// TIA Portal V17 export
// export: Created 2023-02-14T02:49:31.6771521Z, ExportSetting WithDefaults, DisplayName Totally Integrated Automation Portal, DisplayVersion V17, DisplayName TIA Portal Openness, DisplayVersion V17, DisplayName TIA Portal Teamcenter Gateway, DisplayVersion V17, DisplayName TIA Portal Version Control Interface, DisplayVersion V17, DisplayName SINAMICS Startdrive Advanced, DisplayVersion V17, DisplayName SINAMICS Startdrive G130, G150, S120, S150, SINAMICS MV, S210, DisplayVersion V17, DisplayName SINAMICS Startdrive G110M, G120, G120C, G120D, G120P, G115D, DisplayVersion V17, DisplayName STEP 7 Professional, DisplayVersion V17, DisplayName STEP 7 Safety, DisplayVersion V17, DisplayName WinCC Professional, DisplayVersion V17
FUNCTION_BLOCK "IO Motor MCC Preparation"   // FB15, LAD
{ S7_Optimized_Access := 'FALSE' }
VERSION : 0.1
// stored: AutoNumber true, IsIECCheckEnabled false, SetENOAutomatically false, UDAEnableTagReadback false
   VAR_INPUT
      lock : Bool;
      Init : Bool;
      EM_Stop : Bool;
      Testing : Bool;
      Reset : Bool;
   END_VAR
   VAR
      "P-01.01" { S7_SetPoint := 'True'} : "Motor_w_VSD";
      "P-02.01" { S7_SetPoint := 'True'} : "Motor_w_VSD";
      "P-02.03" { S7_SetPoint := 'True'} : "Motor_w_VSD";
      "P-03.01" { S7_SetPoint := 'True'} : "Motor_w_VSD";
      "P-03.03" { S7_SetPoint := 'True'} : "Motor_w_VSD";
      "P-04.01" { S7_SetPoint := 'True'} : "Motor_w_VSD";
      "XA-05.01" { S7_SetPoint := 'True'} : "Motor_w_VSD";
      "P-05.01" { S7_SetPoint := 'True'} : "Motor_w_VSD";
      "P-05.03_DOL" { S7_SetPoint := 'True'} : "Motor";
      "P-06.01" { S7_SetPoint := 'True'} : "Motor_w_VSD";
      "P-07.01" { S7_SetPoint := 'True'} : "Motor_w_VSD";
      "P-08.01" { S7_SetPoint := 'True'} : "Motor_w_VSD";
      "P-08.02" { S7_SetPoint := 'True'} : "Motor_w_VSD";
      "XA-09.01" { S7_SetPoint := 'True'} : "Motor_w_VSD";
      "P-09.01" { S7_SetPoint := 'True'} : "Motor_w_VSD";
      "P-09.03" { S7_SetPoint := 'True'} : "Motor";
      "P-10.01" { S7_SetPoint := 'True'} : "Motor_w_VSD";
      "P-51.01" { S7_SetPoint := 'True'} : "Motor_w_VSD";
   END_VAR
BEGIN

REGION Network 1: Testing
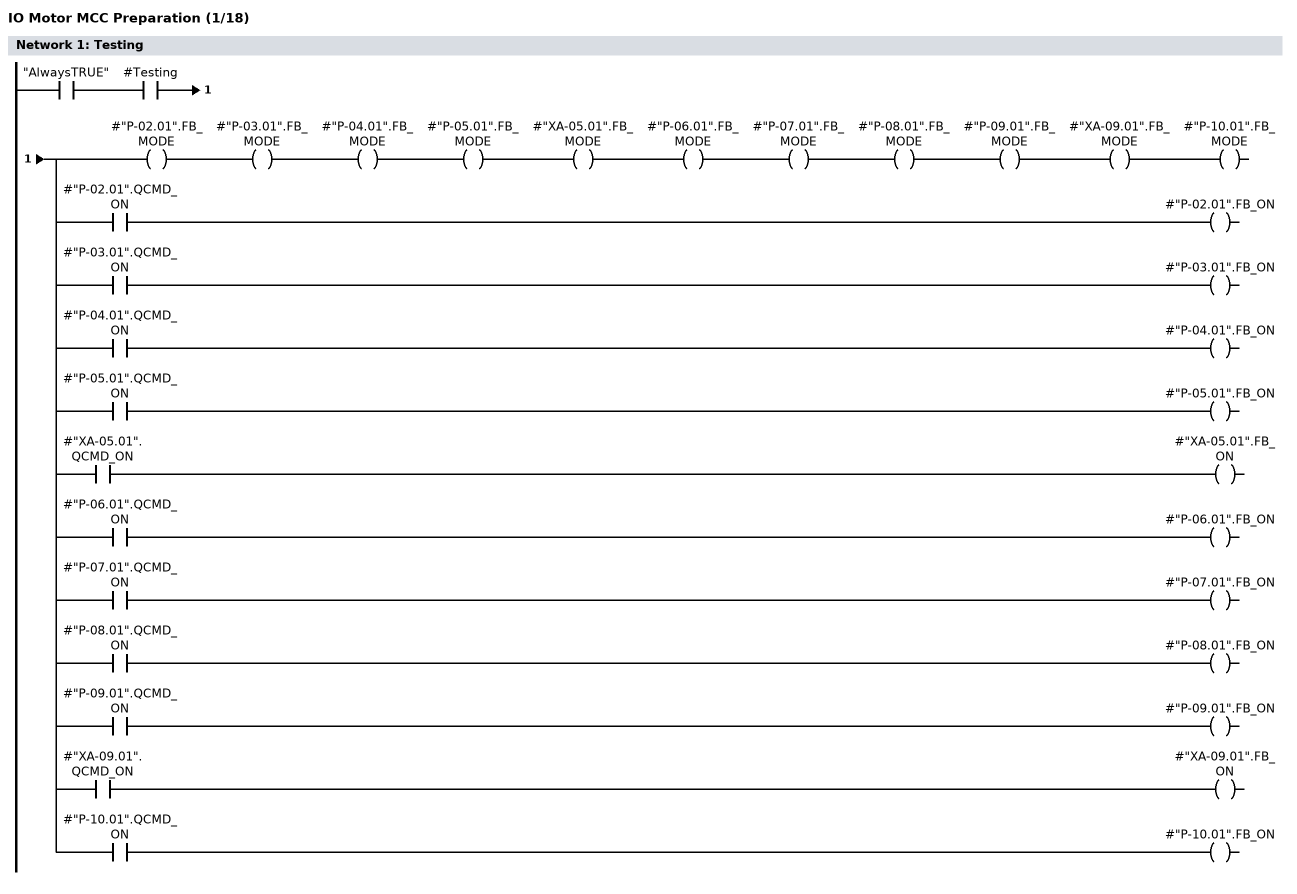
   RUNG wire#powerrail
      Contact( "AlwaysTRUE" )
      Contact( #Testing )
      wire#w1
      Coil( #"P-02.01".FB_MODE )
      Coil( #"P-03.01".FB_MODE )
      Coil( #"P-04.01".FB_MODE )
      Coil( #"P-05.01".FB_MODE )
      Coil( #"XA-05.01".FB_MODE )
      Coil( #"P-06.01".FB_MODE )
      Coil( #"P-07.01".FB_MODE )
      Coil( #"P-08.01".FB_MODE )
      Coil( #"P-09.01".FB_MODE )
      Coil( #"XA-09.01".FB_MODE )
      Coil( #"P-10.01".FB_MODE )
   END_RUNG
   RUNG wire#w1
      Contact( #"P-02.01".QCMD_ON )
      Coil( #"P-02.01".FB_ON )
   END_RUNG
   RUNG wire#w1
      Contact( #"P-03.01".QCMD_ON )
      Coil( #"P-03.01".FB_ON )
   END_RUNG
   RUNG wire#w1
      Contact( #"P-04.01".QCMD_ON )
      Coil( #"P-04.01".FB_ON )
   END_RUNG
   RUNG wire#w1
      Contact( #"P-05.01".QCMD_ON )
      Coil( #"P-05.01".FB_ON )
   END_RUNG
   RUNG wire#w1
      Contact( #"XA-05.01".QCMD_ON )
      Coil( #"XA-05.01".FB_ON )
   END_RUNG
   RUNG wire#w1
      Contact( #"P-06.01".QCMD_ON )
      Coil( #"P-06.01".FB_ON )
   END_RUNG
   RUNG wire#w1
      Contact( #"P-07.01".QCMD_ON )
      Coil( #"P-07.01".FB_ON )
   END_RUNG
   RUNG wire#w1
      Contact( #"P-08.01".QCMD_ON )
      Coil( #"P-08.01".FB_ON )
   END_RUNG
   RUNG wire#w1
      Contact( #"P-09.01".QCMD_ON )
      Coil( #"P-09.01".FB_ON )
   END_RUNG
   RUNG wire#w1
      Contact( #"XA-09.01".QCMD_ON )
      Coil( #"XA-09.01".FB_ON )
   END_RUNG
   RUNG wire#w1
      Contact( #"P-10.01".QCMD_ON )
      Coil( #"P-10.01".FB_ON )
   END_RUNG
   // the same network as SCL:
   #"P-02.01".FB_MODE := "AlwaysTRUE" AND #Testing;
   #"P-03.01".FB_MODE := #"P-02.01".FB_MODE;
   #"P-04.01".FB_MODE := #"P-02.01".FB_MODE;
   #"P-05.01".FB_MODE := #"P-02.01".FB_MODE;
   #"XA-05.01".FB_MODE := #"P-02.01".FB_MODE;
   #"P-06.01".FB_MODE := #"P-02.01".FB_MODE;
   #"P-07.01".FB_MODE := #"P-02.01".FB_MODE;
   #"P-08.01".FB_MODE := #"P-02.01".FB_MODE;
   #"P-09.01".FB_MODE := #"P-02.01".FB_MODE;
   #"XA-09.01".FB_MODE := #"P-02.01".FB_MODE;
   #"P-10.01".FB_MODE := #"P-02.01".FB_MODE;
   #"P-02.01".FB_ON := #"P-02.01".FB_MODE AND #"P-02.01".QCMD_ON;
   #"P-03.01".FB_ON := #"P-02.01".FB_MODE AND #"P-03.01".QCMD_ON;
   #"P-04.01".FB_ON := #"P-02.01".FB_MODE AND #"P-04.01".QCMD_ON;
   #"P-05.01".FB_ON := #"P-02.01".FB_MODE AND #"P-05.01".QCMD_ON;
   #"XA-05.01".FB_ON := #"P-02.01".FB_MODE AND #"XA-05.01".QCMD_ON;
   #"P-06.01".FB_ON := #"P-02.01".FB_MODE AND #"P-06.01".QCMD_ON;
   #"P-07.01".FB_ON := #"P-02.01".FB_MODE AND #"P-07.01".QCMD_ON;
   #"P-08.01".FB_ON := #"P-02.01".FB_MODE AND #"P-08.01".QCMD_ON;
   #"P-09.01".FB_ON := #"P-02.01".FB_MODE AND #"P-09.01".QCMD_ON;
   #"XA-09.01".FB_ON := #"P-02.01".FB_MODE AND #"XA-09.01".QCMD_ON;
   #"P-10.01".FB_ON := #"P-02.01".FB_MODE AND #"P-10.01".QCMD_ON;
END_REGION

REGION Network 2: P-02.01
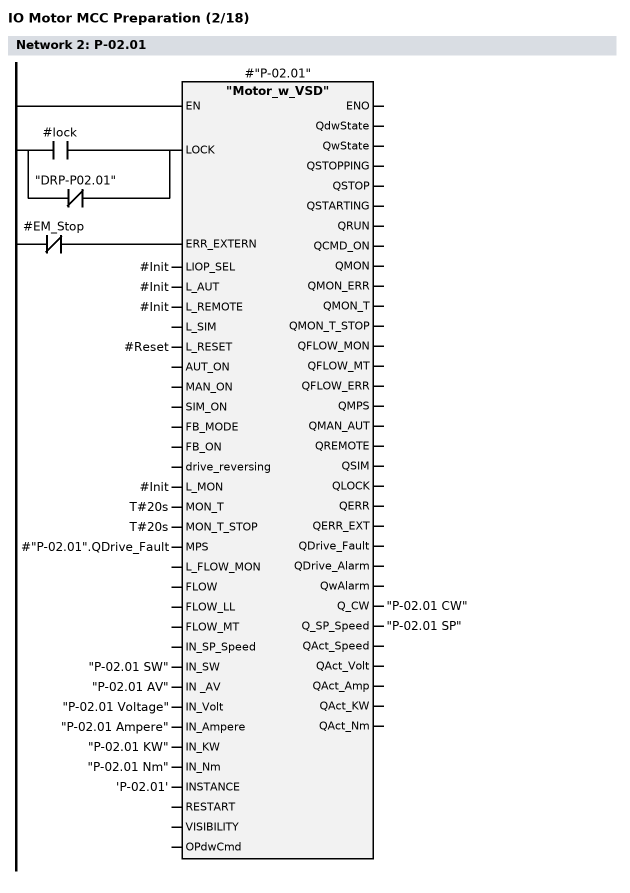
   RUNG wire#powerrail
      #"P-02.01"(LOCK := wire#w1, ERR_EXTERN := wire#w2, LIOP_SEL := #Init, L_AUT := #Init, L_REMOTE := #Init, L_SIM :=, L_RESET := #Reset, AUT_ON :=, MAN_ON :=, SIM_ON :=, FB_MODE :=, FB_ON :=, drive_reversing :=, L_MON := #Init, MON_T := T#20s, MON_T_STOP := T#20s, MPS := #"P-02.01".QDrive_Fault, L_FLOW_MON :=, FLOW :=, FLOW_LL :=, FLOW_MT :=, IN_SP_Speed :=, IN_SW := "P-02.01 SW", "IN _AV" := "P-02.01 AV", IN_Volt := "P-02.01 Voltage", IN_Ampere := "P-02.01 Ampere", IN_KW := "P-02.01 KW", IN_Nm := "P-02.01 Nm", INSTANCE := 'P-02.01', RESTART :=, VISIBILITY :=, OPdwCmd :=, QdwState =>, QwState =>, QSTOPPING =>, QSTOP =>, QSTARTING =>, QRUN =>, QCMD_ON =>, QMON =>, QMON_ERR =>, QMON_T =>, QMON_T_STOP =>, QFLOW_MON =>, QFLOW_MT =>, QFLOW_ERR =>, QMPS =>, QMAN_AUT =>, QREMOTE =>, QSIM =>, QLOCK =>, QERR =>, QERR_EXT =>, QDrive_Fault =>, QDrive_Alarm =>, QwAlarm =>, Q_CW => "P-02.01 CW", Q_SP_Speed => "P-02.01 SP", QAct_Speed =>, QAct_Volt =>, QAct_Amp =>, QAct_KW =>, QAct_Nm =>)
   END_RUNG
   RUNG wire#powerrail
      Contact( #lock )
   END_RUNG wire#w1
   RUNG wire#powerrail
      I_Contact( "DRP-P02.01" )
   END_RUNG wire#w1
   RUNG wire#powerrail
      I_Contact( #EM_Stop )
   END_RUNG wire#w2
   // the same network as SCL:
   #"P-02.01"(LOCK := #lock OR NOT "DRP-P02.01",   // "Motor_w_VSD"
              ERR_EXTERN := NOT #EM_Stop,
              LIOP_SEL := #Init,
              L_AUT := #Init,
              L_REMOTE := #Init,
              L_RESET := #Reset,
              L_MON := #Init,
              MON_T := T#20s,
              MON_T_STOP := T#20s,
              MPS := #"P-02.01".QDrive_Fault,
              IN_SW := "P-02.01 SW",
              "IN _AV" := "P-02.01 AV",
              IN_Volt := "P-02.01 Voltage",
              IN_Ampere := "P-02.01 Ampere",
              IN_KW := "P-02.01 KW",
              IN_Nm := "P-02.01 Nm",
              INSTANCE := 'P-02.01',
              Q_CW => "P-02.01 CW",
              Q_SP_Speed => "P-02.01 SP");
END_REGION

REGION Network 3: P-02.03
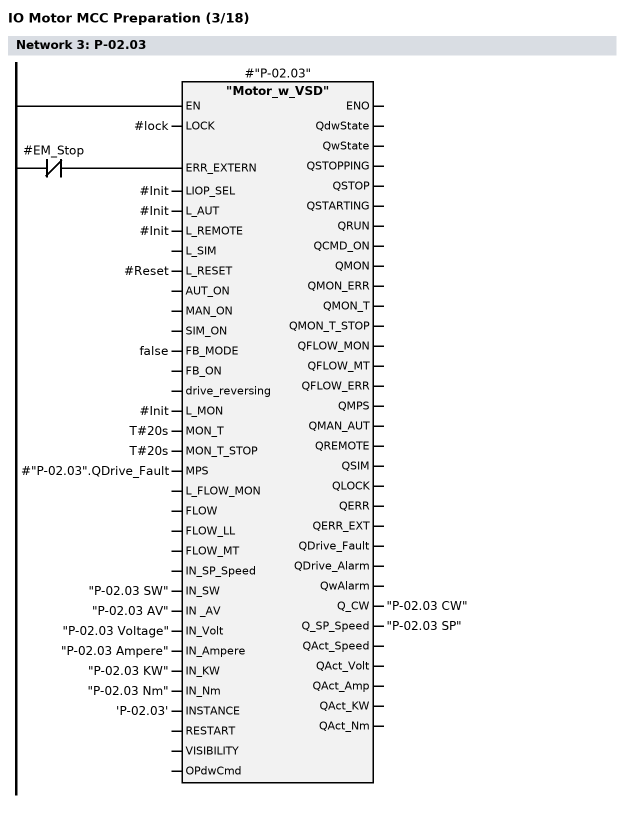
   RUNG wire#powerrail
      #"P-02.03"(ERR_EXTERN := wire#w1, LOCK := #lock, LIOP_SEL := #Init, L_AUT := #Init, L_REMOTE := #Init, L_SIM :=, L_RESET := #Reset, AUT_ON :=, MAN_ON :=, SIM_ON :=, FB_MODE := false, FB_ON :=, drive_reversing :=, L_MON := #Init, MON_T := T#20s, MON_T_STOP := T#20s, MPS := #"P-02.03".QDrive_Fault, L_FLOW_MON :=, FLOW :=, FLOW_LL :=, FLOW_MT :=, IN_SP_Speed :=, IN_SW := "P-02.03 SW", "IN _AV" := "P-02.03 AV", IN_Volt := "P-02.03 Voltage", IN_Ampere := "P-02.03 Ampere", IN_KW := "P-02.03 KW", IN_Nm := "P-02.03 Nm", INSTANCE := 'P-02.03', RESTART :=, VISIBILITY :=, OPdwCmd :=, QdwState =>, QwState =>, QSTOPPING =>, QSTOP =>, QSTARTING =>, QRUN =>, QCMD_ON =>, QMON =>, QMON_ERR =>, QMON_T =>, QMON_T_STOP =>, QFLOW_MON =>, QFLOW_MT =>, QFLOW_ERR =>, QMPS =>, QMAN_AUT =>, QREMOTE =>, QSIM =>, QLOCK =>, QERR =>, QERR_EXT =>, QDrive_Fault =>, QDrive_Alarm =>, QwAlarm =>, Q_CW => "P-02.03 CW", Q_SP_Speed => "P-02.03 SP", QAct_Speed =>, QAct_Volt =>, QAct_Amp =>, QAct_KW =>, QAct_Nm =>)
   END_RUNG
   RUNG wire#powerrail
      I_Contact( #EM_Stop )
   END_RUNG wire#w1
   // the same network as SCL:
   #"P-02.03"(LOCK := #lock,   // "Motor_w_VSD"
              ERR_EXTERN := NOT #EM_Stop,
              LIOP_SEL := #Init,
              L_AUT := #Init,
              L_REMOTE := #Init,
              L_RESET := #Reset,
              FB_MODE := false,
              L_MON := #Init,
              MON_T := T#20s,
              MON_T_STOP := T#20s,
              MPS := #"P-02.03".QDrive_Fault,
              IN_SW := "P-02.03 SW",
              "IN _AV" := "P-02.03 AV",
              IN_Volt := "P-02.03 Voltage",
              IN_Ampere := "P-02.03 Ampere",
              IN_KW := "P-02.03 KW",
              IN_Nm := "P-02.03 Nm",
              INSTANCE := 'P-02.03',
              Q_CW => "P-02.03 CW",
              Q_SP_Speed => "P-02.03 SP");
END_REGION

REGION Network 4: P-03.01
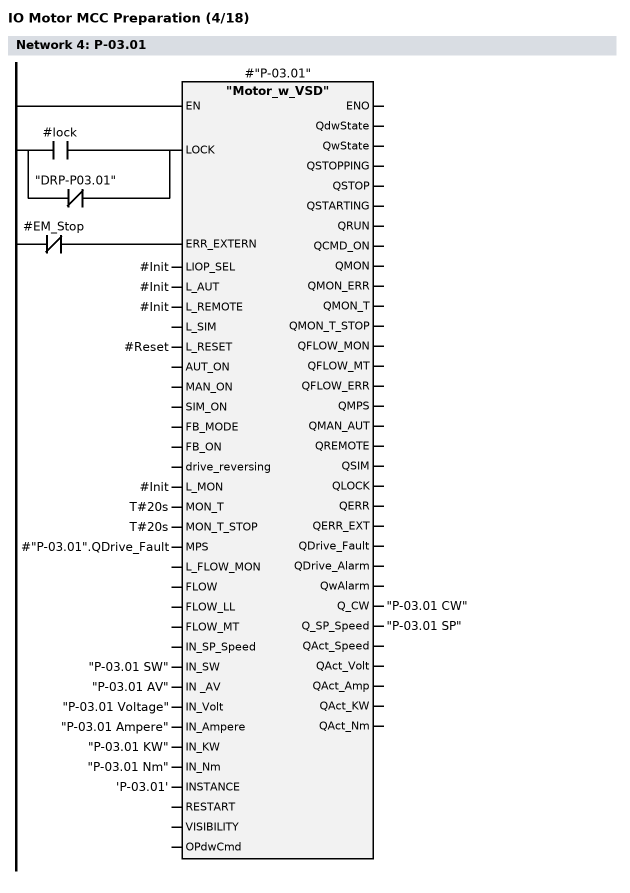
   RUNG wire#powerrail
      #"P-03.01"(LOCK := wire#w1, ERR_EXTERN := wire#w2, LIOP_SEL := #Init, L_AUT := #Init, L_REMOTE := #Init, L_SIM :=, L_RESET := #Reset, AUT_ON :=, MAN_ON :=, SIM_ON :=, FB_MODE :=, FB_ON :=, drive_reversing :=, L_MON := #Init, MON_T := T#20s, MON_T_STOP := T#20s, MPS := #"P-03.01".QDrive_Fault, L_FLOW_MON :=, FLOW :=, FLOW_LL :=, FLOW_MT :=, IN_SP_Speed :=, IN_SW := "P-03.01 SW", "IN _AV" := "P-03.01 AV", IN_Volt := "P-03.01 Voltage", IN_Ampere := "P-03.01 Ampere", IN_KW := "P-03.01 KW", IN_Nm := "P-03.01 Nm", INSTANCE := 'P-03.01', RESTART :=, VISIBILITY :=, OPdwCmd :=, QdwState =>, QwState =>, QSTOPPING =>, QSTOP =>, QSTARTING =>, QRUN =>, QCMD_ON =>, QMON =>, QMON_ERR =>, QMON_T =>, QMON_T_STOP =>, QFLOW_MON =>, QFLOW_MT =>, QFLOW_ERR =>, QMPS =>, QMAN_AUT =>, QREMOTE =>, QSIM =>, QLOCK =>, QERR =>, QERR_EXT =>, QDrive_Fault =>, QDrive_Alarm =>, QwAlarm =>, Q_CW => "P-03.01 CW", Q_SP_Speed => "P-03.01 SP", QAct_Speed =>, QAct_Volt =>, QAct_Amp =>, QAct_KW =>, QAct_Nm =>)
   END_RUNG
   RUNG wire#powerrail
      Contact( #lock )
   END_RUNG wire#w1
   RUNG wire#powerrail
      I_Contact( "DRP-P03.01" )
   END_RUNG wire#w1
   RUNG wire#powerrail
      I_Contact( #EM_Stop )
   END_RUNG wire#w2
   // the same network as SCL:
   #"P-03.01"(LOCK := #lock OR NOT "DRP-P03.01",   // "Motor_w_VSD"
              ERR_EXTERN := NOT #EM_Stop,
              LIOP_SEL := #Init,
              L_AUT := #Init,
              L_REMOTE := #Init,
              L_RESET := #Reset,
              L_MON := #Init,
              MON_T := T#20s,
              MON_T_STOP := T#20s,
              MPS := #"P-03.01".QDrive_Fault,
              IN_SW := "P-03.01 SW",
              "IN _AV" := "P-03.01 AV",
              IN_Volt := "P-03.01 Voltage",
              IN_Ampere := "P-03.01 Ampere",
              IN_KW := "P-03.01 KW",
              IN_Nm := "P-03.01 Nm",
              INSTANCE := 'P-03.01',
              Q_CW => "P-03.01 CW",
              Q_SP_Speed => "P-03.01 SP");
END_REGION

REGION Network 5: P-03.03
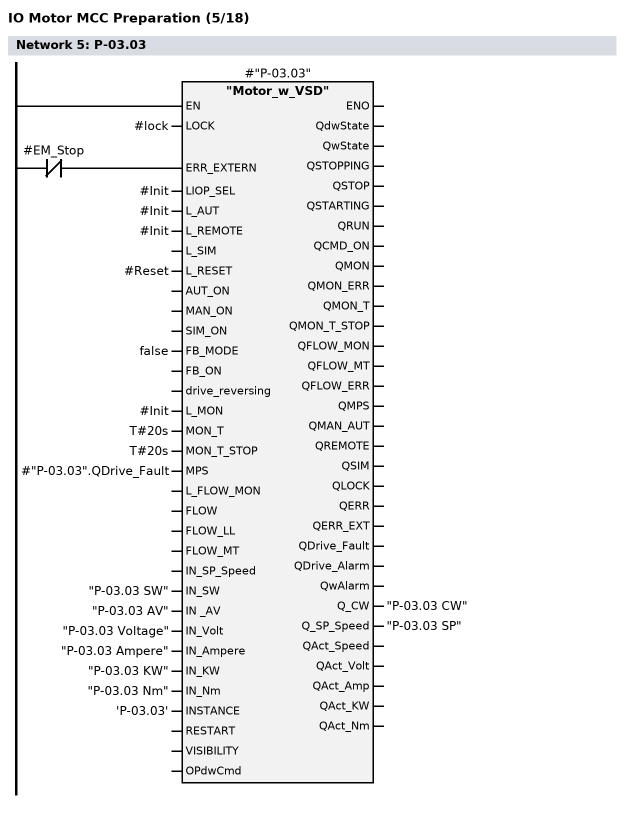
   RUNG wire#powerrail
      #"P-03.03"(ERR_EXTERN := wire#w1, LOCK := #lock, LIOP_SEL := #Init, L_AUT := #Init, L_REMOTE := #Init, L_SIM :=, L_RESET := #Reset, AUT_ON :=, MAN_ON :=, SIM_ON :=, FB_MODE := false, FB_ON :=, drive_reversing :=, L_MON := #Init, MON_T := T#20s, MON_T_STOP := T#20s, MPS := #"P-03.03".QDrive_Fault, L_FLOW_MON :=, FLOW :=, FLOW_LL :=, FLOW_MT :=, IN_SP_Speed :=, IN_SW := "P-03.03 SW", "IN _AV" := "P-03.03 AV", IN_Volt := "P-03.03 Voltage", IN_Ampere := "P-03.03 Ampere", IN_KW := "P-03.03 KW", IN_Nm := "P-03.03 Nm", INSTANCE := 'P-03.03', RESTART :=, VISIBILITY :=, OPdwCmd :=, QdwState =>, QwState =>, QSTOPPING =>, QSTOP =>, QSTARTING =>, QRUN =>, QCMD_ON =>, QMON =>, QMON_ERR =>, QMON_T =>, QMON_T_STOP =>, QFLOW_MON =>, QFLOW_MT =>, QFLOW_ERR =>, QMPS =>, QMAN_AUT =>, QREMOTE =>, QSIM =>, QLOCK =>, QERR =>, QERR_EXT =>, QDrive_Fault =>, QDrive_Alarm =>, QwAlarm =>, Q_CW => "P-03.03 CW", Q_SP_Speed => "P-03.03 SP", QAct_Speed =>, QAct_Volt =>, QAct_Amp =>, QAct_KW =>, QAct_Nm =>)
   END_RUNG
   RUNG wire#powerrail
      I_Contact( #EM_Stop )
   END_RUNG wire#w1
   // the same network as SCL:
   #"P-03.03"(LOCK := #lock,   // "Motor_w_VSD"
              ERR_EXTERN := NOT #EM_Stop,
              LIOP_SEL := #Init,
              L_AUT := #Init,
              L_REMOTE := #Init,
              L_RESET := #Reset,
              FB_MODE := false,
              L_MON := #Init,
              MON_T := T#20s,
              MON_T_STOP := T#20s,
              MPS := #"P-03.03".QDrive_Fault,
              IN_SW := "P-03.03 SW",
              "IN _AV" := "P-03.03 AV",
              IN_Volt := "P-03.03 Voltage",
              IN_Ampere := "P-03.03 Ampere",
              IN_KW := "P-03.03 KW",
              IN_Nm := "P-03.03 Nm",
              INSTANCE := 'P-03.03',
              Q_CW => "P-03.03 CW",
              Q_SP_Speed => "P-03.03 SP");
END_REGION

REGION Network 6: P-04.01
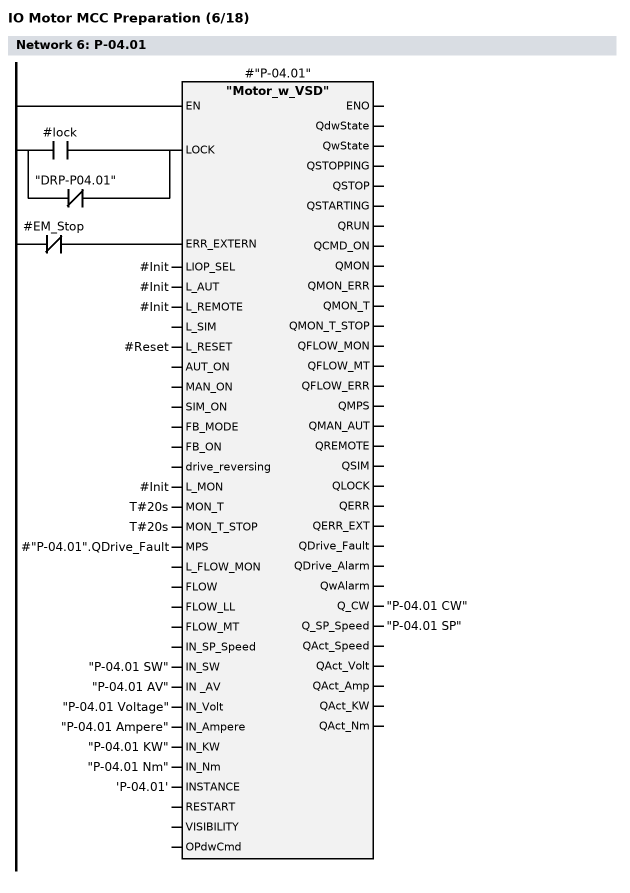
   RUNG wire#powerrail
      #"P-04.01"(LOCK := wire#w1, ERR_EXTERN := wire#w2, LIOP_SEL := #Init, L_AUT := #Init, L_REMOTE := #Init, L_SIM :=, L_RESET := #Reset, AUT_ON :=, MAN_ON :=, SIM_ON :=, FB_MODE :=, FB_ON :=, drive_reversing :=, L_MON := #Init, MON_T := T#20s, MON_T_STOP := T#20s, MPS := #"P-04.01".QDrive_Fault, L_FLOW_MON :=, FLOW :=, FLOW_LL :=, FLOW_MT :=, IN_SP_Speed :=, IN_SW := "P-04.01 SW", "IN _AV" := "P-04.01 AV", IN_Volt := "P-04.01 Voltage", IN_Ampere := "P-04.01 Ampere", IN_KW := "P-04.01 KW", IN_Nm := "P-04.01 Nm", INSTANCE := 'P-04.01', RESTART :=, VISIBILITY :=, OPdwCmd :=, QdwState =>, QwState =>, QSTOPPING =>, QSTOP =>, QSTARTING =>, QRUN =>, QCMD_ON =>, QMON =>, QMON_ERR =>, QMON_T =>, QMON_T_STOP =>, QFLOW_MON =>, QFLOW_MT =>, QFLOW_ERR =>, QMPS =>, QMAN_AUT =>, QREMOTE =>, QSIM =>, QLOCK =>, QERR =>, QERR_EXT =>, QDrive_Fault =>, QDrive_Alarm =>, QwAlarm =>, Q_CW => "P-04.01 CW", Q_SP_Speed => "P-04.01 SP", QAct_Speed =>, QAct_Volt =>, QAct_Amp =>, QAct_KW =>, QAct_Nm =>)
   END_RUNG
   RUNG wire#powerrail
      Contact( #lock )
   END_RUNG wire#w1
   RUNG wire#powerrail
      I_Contact( "DRP-P04.01" )
   END_RUNG wire#w1
   RUNG wire#powerrail
      I_Contact( #EM_Stop )
   END_RUNG wire#w2
   // the same network as SCL:
   #"P-04.01"(LOCK := #lock OR NOT "DRP-P04.01",   // "Motor_w_VSD"
              ERR_EXTERN := NOT #EM_Stop,
              LIOP_SEL := #Init,
              L_AUT := #Init,
              L_REMOTE := #Init,
              L_RESET := #Reset,
              L_MON := #Init,
              MON_T := T#20s,
              MON_T_STOP := T#20s,
              MPS := #"P-04.01".QDrive_Fault,
              IN_SW := "P-04.01 SW",
              "IN _AV" := "P-04.01 AV",
              IN_Volt := "P-04.01 Voltage",
              IN_Ampere := "P-04.01 Ampere",
              IN_KW := "P-04.01 KW",
              IN_Nm := "P-04.01 Nm",
              INSTANCE := 'P-04.01',
              Q_CW => "P-04.01 CW",
              Q_SP_Speed => "P-04.01 SP");
END_REGION

REGION Network 7: XA-05.01
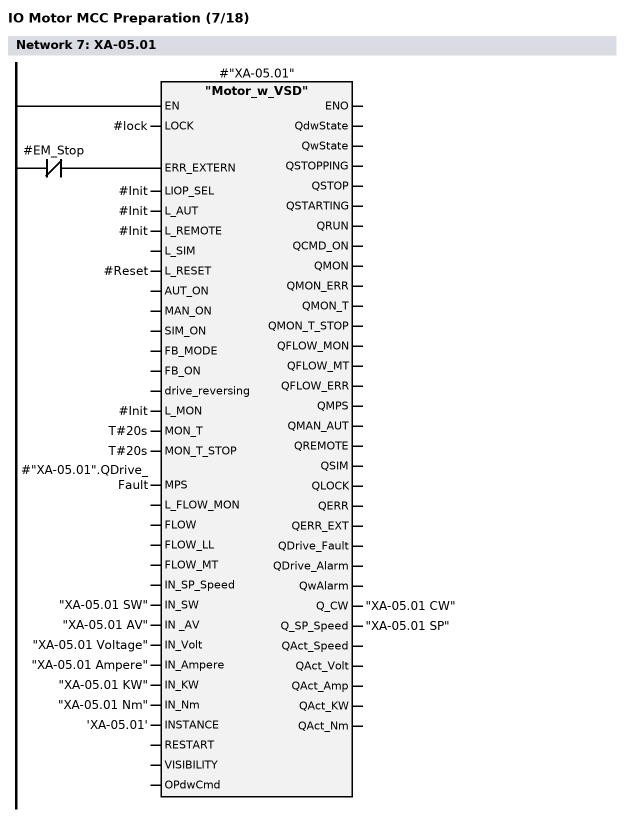
   RUNG wire#powerrail
      #"XA-05.01"(ERR_EXTERN := wire#w1, LOCK := #lock, LIOP_SEL := #Init, L_AUT := #Init, L_REMOTE := #Init, L_SIM :=, L_RESET := #Reset, AUT_ON :=, MAN_ON :=, SIM_ON :=, FB_MODE :=, FB_ON :=, drive_reversing :=, L_MON := #Init, MON_T := T#20s, MON_T_STOP := T#20s, MPS := #"XA-05.01".QDrive_Fault, L_FLOW_MON :=, FLOW :=, FLOW_LL :=, FLOW_MT :=, IN_SP_Speed :=, IN_SW := "XA-05.01 SW", "IN _AV" := "XA-05.01 AV", IN_Volt := "XA-05.01 Voltage", IN_Ampere := "XA-05.01 Ampere", IN_KW := "XA-05.01 KW", IN_Nm := "XA-05.01 Nm", INSTANCE := 'XA-05.01', RESTART :=, VISIBILITY :=, OPdwCmd :=, QdwState =>, QwState =>, QSTOPPING =>, QSTOP =>, QSTARTING =>, QRUN =>, QCMD_ON =>, QMON =>, QMON_ERR =>, QMON_T =>, QMON_T_STOP =>, QFLOW_MON =>, QFLOW_MT =>, QFLOW_ERR =>, QMPS =>, QMAN_AUT =>, QREMOTE =>, QSIM =>, QLOCK =>, QERR =>, QERR_EXT =>, QDrive_Fault =>, QDrive_Alarm =>, QwAlarm =>, Q_CW => "XA-05.01 CW", Q_SP_Speed => "XA-05.01 SP", QAct_Speed =>, QAct_Volt =>, QAct_Amp =>, QAct_KW =>, QAct_Nm =>)
   END_RUNG
   RUNG wire#powerrail
      I_Contact( #EM_Stop )
   END_RUNG wire#w1
   // the same network as SCL:
   #"XA-05.01"(LOCK := #lock,   // "Motor_w_VSD"
               ERR_EXTERN := NOT #EM_Stop,
               LIOP_SEL := #Init,
               L_AUT := #Init,
               L_REMOTE := #Init,
               L_RESET := #Reset,
               L_MON := #Init,
               MON_T := T#20s,
               MON_T_STOP := T#20s,
               MPS := #"XA-05.01".QDrive_Fault,
               IN_SW := "XA-05.01 SW",
               "IN _AV" := "XA-05.01 AV",
               IN_Volt := "XA-05.01 Voltage",
               IN_Ampere := "XA-05.01 Ampere",
               IN_KW := "XA-05.01 KW",
               IN_Nm := "XA-05.01 Nm",
               INSTANCE := 'XA-05.01',
               Q_CW => "XA-05.01 CW",
               Q_SP_Speed => "XA-05.01 SP");
END_REGION

REGION Network 8: P-05.01
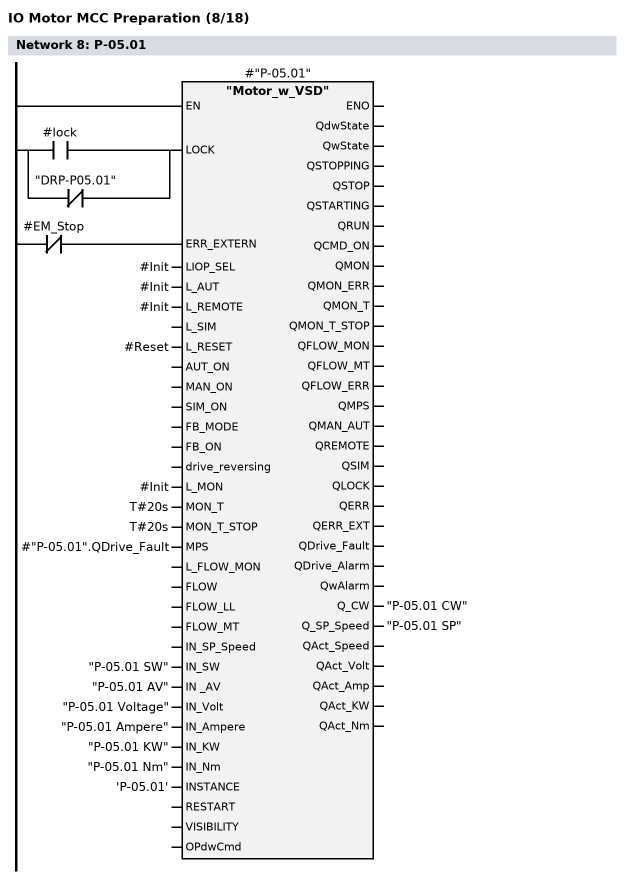
   RUNG wire#powerrail
      #"P-05.01"(LOCK := wire#w1, ERR_EXTERN := wire#w2, LIOP_SEL := #Init, L_AUT := #Init, L_REMOTE := #Init, L_SIM :=, L_RESET := #Reset, AUT_ON :=, MAN_ON :=, SIM_ON :=, FB_MODE :=, FB_ON :=, drive_reversing :=, L_MON := #Init, MON_T := T#20s, MON_T_STOP := T#20s, MPS := #"P-05.01".QDrive_Fault, L_FLOW_MON :=, FLOW :=, FLOW_LL :=, FLOW_MT :=, IN_SP_Speed :=, IN_SW := "P-05.01 SW", "IN _AV" := "P-05.01 AV", IN_Volt := "P-05.01 Voltage", IN_Ampere := "P-05.01 Ampere", IN_KW := "P-05.01 KW", IN_Nm := "P-05.01 Nm", INSTANCE := 'P-05.01', RESTART :=, VISIBILITY :=, OPdwCmd :=, QdwState =>, QwState =>, QSTOPPING =>, QSTOP =>, QSTARTING =>, QRUN =>, QCMD_ON =>, QMON =>, QMON_ERR =>, QMON_T =>, QMON_T_STOP =>, QFLOW_MON =>, QFLOW_MT =>, QFLOW_ERR =>, QMPS =>, QMAN_AUT =>, QREMOTE =>, QSIM =>, QLOCK =>, QERR =>, QERR_EXT =>, QDrive_Fault =>, QDrive_Alarm =>, QwAlarm =>, Q_CW => "P-05.01 CW", Q_SP_Speed => "P-05.01 SP", QAct_Speed =>, QAct_Volt =>, QAct_Amp =>, QAct_KW =>, QAct_Nm =>)
   END_RUNG
   RUNG wire#powerrail
      Contact( #lock )
   END_RUNG wire#w1
   RUNG wire#powerrail
      I_Contact( "DRP-P05.01" )
   END_RUNG wire#w1
   RUNG wire#powerrail
      I_Contact( #EM_Stop )
   END_RUNG wire#w2
   // the same network as SCL:
   #"P-05.01"(LOCK := #lock OR NOT "DRP-P05.01",   // "Motor_w_VSD"
              ERR_EXTERN := NOT #EM_Stop,
              LIOP_SEL := #Init,
              L_AUT := #Init,
              L_REMOTE := #Init,
              L_RESET := #Reset,
              L_MON := #Init,
              MON_T := T#20s,
              MON_T_STOP := T#20s,
              MPS := #"P-05.01".QDrive_Fault,
              IN_SW := "P-05.01 SW",
              "IN _AV" := "P-05.01 AV",
              IN_Volt := "P-05.01 Voltage",
              IN_Ampere := "P-05.01 Ampere",
              IN_KW := "P-05.01 KW",
              IN_Nm := "P-05.01 Nm",
              INSTANCE := 'P-05.01',
              Q_CW => "P-05.01 CW",
              Q_SP_Speed => "P-05.01 SP");
END_REGION

REGION Network 9: P-05.03 DOL
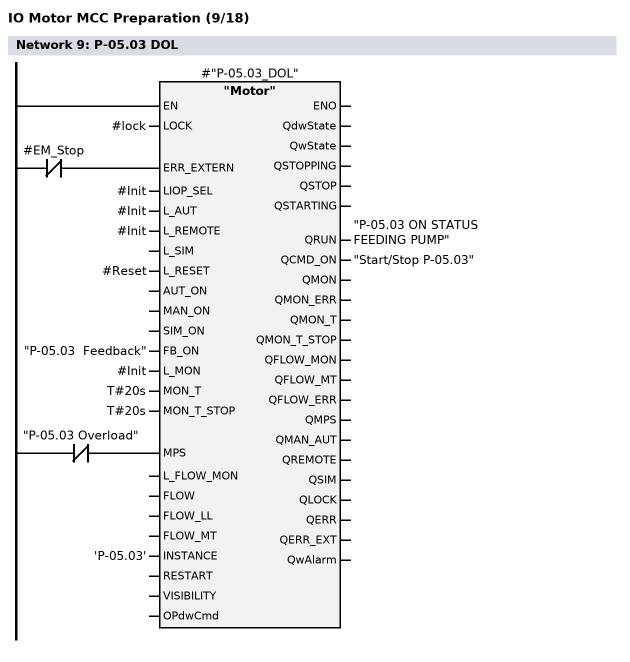
   RUNG wire#powerrail
      #"P-05.03_DOL"(ERR_EXTERN := wire#w1, MPS := wire#w2, LOCK := #lock, LIOP_SEL := #Init, L_AUT := #Init, L_REMOTE := #Init, L_SIM :=, L_RESET := #Reset, AUT_ON :=, MAN_ON :=, SIM_ON :=, FB_ON := "P-05.03  Feedback", L_MON := #Init, MON_T := T#20s, MON_T_STOP := T#20s, L_FLOW_MON :=, FLOW :=, FLOW_LL :=, FLOW_MT :=, INSTANCE := 'P-05.03', RESTART :=, VISIBILITY :=, OPdwCmd :=, QdwState =>, QwState =>, QSTOPPING =>, QSTOP =>, QSTARTING =>, QRUN => "P-05.03 ON STATUS FEEDING PUMP", QCMD_ON => "Start/Stop P-05.03", QMON =>, QMON_ERR =>, QMON_T =>, QMON_T_STOP =>, QFLOW_MON =>, QFLOW_MT =>, QFLOW_ERR =>, QMPS =>, QMAN_AUT =>, QREMOTE =>, QSIM =>, QLOCK =>, QERR =>, QERR_EXT =>, QwAlarm =>)
   END_RUNG
   RUNG wire#powerrail
      I_Contact( #EM_Stop )
   END_RUNG wire#w1
   RUNG wire#powerrail
      I_Contact( "P-05.03 Overload" )
   END_RUNG wire#w2
   // the same network as SCL:
   #"P-05.03_DOL"(LOCK := #lock,   // "Motor"
                  ERR_EXTERN := NOT #EM_Stop,
                  LIOP_SEL := #Init,
                  L_AUT := #Init,
                  L_REMOTE := #Init,
                  L_RESET := #Reset,
                  FB_ON := "P-05.03  Feedback",
                  L_MON := #Init,
                  MON_T := T#20s,
                  MON_T_STOP := T#20s,
                  MPS := NOT "P-05.03 Overload",
                  INSTANCE := 'P-05.03',
                  QRUN => "P-05.03 ON STATUS FEEDING PUMP",
                  QCMD_ON => "Start/Stop P-05.03");
END_REGION

REGION Network 10: P-06.01
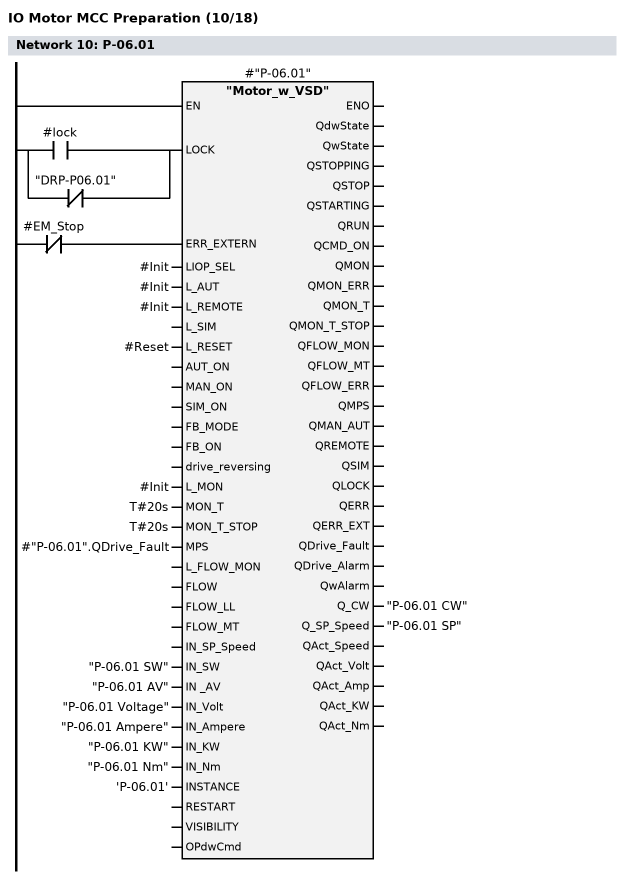
   RUNG wire#powerrail
      #"P-06.01"(LOCK := wire#w1, ERR_EXTERN := wire#w2, LIOP_SEL := #Init, L_AUT := #Init, L_REMOTE := #Init, L_SIM :=, L_RESET := #Reset, AUT_ON :=, MAN_ON :=, SIM_ON :=, FB_MODE :=, FB_ON :=, drive_reversing :=, L_MON := #Init, MON_T := T#20s, MON_T_STOP := T#20s, MPS := #"P-06.01".QDrive_Fault, L_FLOW_MON :=, FLOW :=, FLOW_LL :=, FLOW_MT :=, IN_SP_Speed :=, IN_SW := "P-06.01 SW", "IN _AV" := "P-06.01 AV", IN_Volt := "P-06.01 Voltage", IN_Ampere := "P-06.01 Ampere", IN_KW := "P-06.01 KW", IN_Nm := "P-06.01 Nm", INSTANCE := 'P-06.01', RESTART :=, VISIBILITY :=, OPdwCmd :=, QdwState =>, QwState =>, QSTOPPING =>, QSTOP =>, QSTARTING =>, QRUN =>, QCMD_ON =>, QMON =>, QMON_ERR =>, QMON_T =>, QMON_T_STOP =>, QFLOW_MON =>, QFLOW_MT =>, QFLOW_ERR =>, QMPS =>, QMAN_AUT =>, QREMOTE =>, QSIM =>, QLOCK =>, QERR =>, QERR_EXT =>, QDrive_Fault =>, QDrive_Alarm =>, QwAlarm =>, Q_CW => "P-06.01 CW", Q_SP_Speed => "P-06.01 SP", QAct_Speed =>, QAct_Volt =>, QAct_Amp =>, QAct_KW =>, QAct_Nm =>)
   END_RUNG
   RUNG wire#powerrail
      Contact( #lock )
   END_RUNG wire#w1
   RUNG wire#powerrail
      I_Contact( "DRP-P06.01" )
   END_RUNG wire#w1
   RUNG wire#powerrail
      I_Contact( #EM_Stop )
   END_RUNG wire#w2
   // the same network as SCL:
   #"P-06.01"(LOCK := #lock OR NOT "DRP-P06.01",   // "Motor_w_VSD"
              ERR_EXTERN := NOT #EM_Stop,
              LIOP_SEL := #Init,
              L_AUT := #Init,
              L_REMOTE := #Init,
              L_RESET := #Reset,
              L_MON := #Init,
              MON_T := T#20s,
              MON_T_STOP := T#20s,
              MPS := #"P-06.01".QDrive_Fault,
              IN_SW := "P-06.01 SW",
              "IN _AV" := "P-06.01 AV",
              IN_Volt := "P-06.01 Voltage",
              IN_Ampere := "P-06.01 Ampere",
              IN_KW := "P-06.01 KW",
              IN_Nm := "P-06.01 Nm",
              INSTANCE := 'P-06.01',
              Q_CW => "P-06.01 CW",
              Q_SP_Speed => "P-06.01 SP");
END_REGION

REGION Network 11: P-07.01
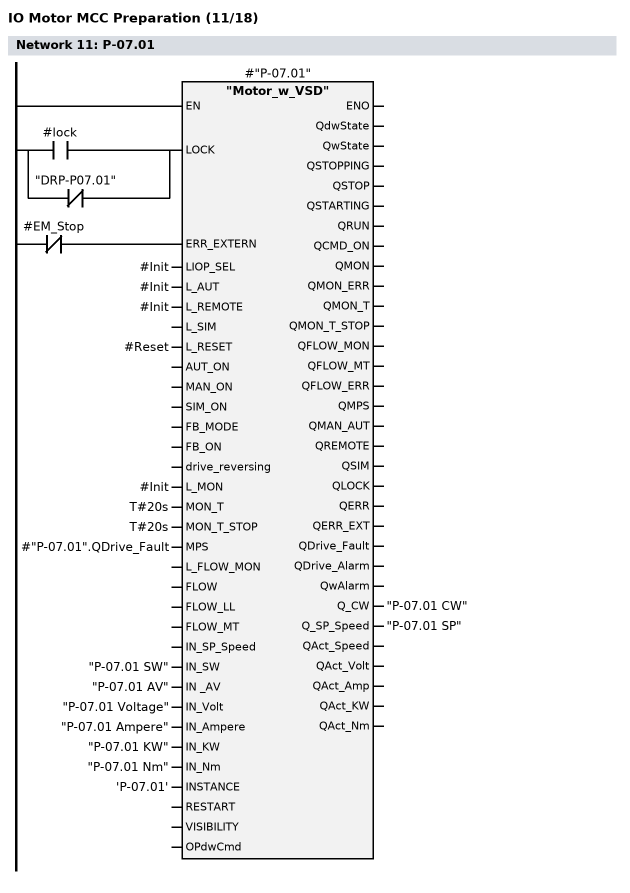
   RUNG wire#powerrail
      #"P-07.01"(LOCK := wire#w1, ERR_EXTERN := wire#w2, LIOP_SEL := #Init, L_AUT := #Init, L_REMOTE := #Init, L_SIM :=, L_RESET := #Reset, AUT_ON :=, MAN_ON :=, SIM_ON :=, FB_MODE :=, FB_ON :=, drive_reversing :=, L_MON := #Init, MON_T := T#20s, MON_T_STOP := T#20s, MPS := #"P-07.01".QDrive_Fault, L_FLOW_MON :=, FLOW :=, FLOW_LL :=, FLOW_MT :=, IN_SP_Speed :=, IN_SW := "P-07.01 SW", "IN _AV" := "P-07.01 AV", IN_Volt := "P-07.01 Voltage", IN_Ampere := "P-07.01 Ampere", IN_KW := "P-07.01 KW", IN_Nm := "P-07.01 Nm", INSTANCE := 'P-07.01', RESTART :=, VISIBILITY :=, OPdwCmd :=, QdwState =>, QwState =>, QSTOPPING =>, QSTOP =>, QSTARTING =>, QRUN =>, QCMD_ON =>, QMON =>, QMON_ERR =>, QMON_T =>, QMON_T_STOP =>, QFLOW_MON =>, QFLOW_MT =>, QFLOW_ERR =>, QMPS =>, QMAN_AUT =>, QREMOTE =>, QSIM =>, QLOCK =>, QERR =>, QERR_EXT =>, QDrive_Fault =>, QDrive_Alarm =>, QwAlarm =>, Q_CW => "P-07.01 CW", Q_SP_Speed => "P-07.01 SP", QAct_Speed =>, QAct_Volt =>, QAct_Amp =>, QAct_KW =>, QAct_Nm =>)
   END_RUNG
   RUNG wire#powerrail
      Contact( #lock )
   END_RUNG wire#w1
   RUNG wire#powerrail
      I_Contact( "DRP-P07.01" )
   END_RUNG wire#w1
   RUNG wire#powerrail
      I_Contact( #EM_Stop )
   END_RUNG wire#w2
   // the same network as SCL:
   #"P-07.01"(LOCK := #lock OR NOT "DRP-P07.01",   // "Motor_w_VSD"
              ERR_EXTERN := NOT #EM_Stop,
              LIOP_SEL := #Init,
              L_AUT := #Init,
              L_REMOTE := #Init,
              L_RESET := #Reset,
              L_MON := #Init,
              MON_T := T#20s,
              MON_T_STOP := T#20s,
              MPS := #"P-07.01".QDrive_Fault,
              IN_SW := "P-07.01 SW",
              "IN _AV" := "P-07.01 AV",
              IN_Volt := "P-07.01 Voltage",
              IN_Ampere := "P-07.01 Ampere",
              IN_KW := "P-07.01 KW",
              IN_Nm := "P-07.01 Nm",
              INSTANCE := 'P-07.01',
              Q_CW => "P-07.01 CW",
              Q_SP_Speed => "P-07.01 SP");
END_REGION

REGION Network 12: P-08.01
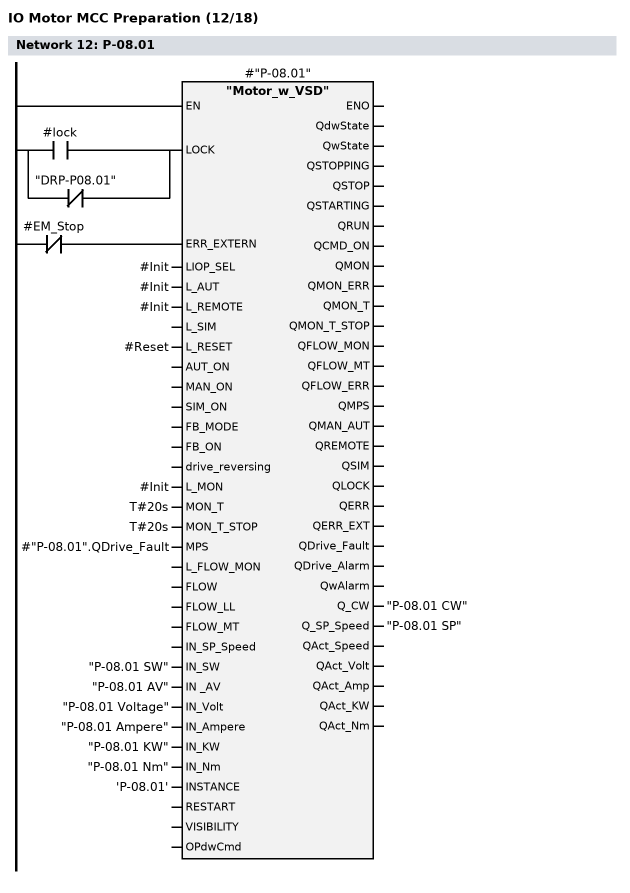
   RUNG wire#powerrail
      #"P-08.01"(LOCK := wire#w1, ERR_EXTERN := wire#w2, LIOP_SEL := #Init, L_AUT := #Init, L_REMOTE := #Init, L_SIM :=, L_RESET := #Reset, AUT_ON :=, MAN_ON :=, SIM_ON :=, FB_MODE :=, FB_ON :=, drive_reversing :=, L_MON := #Init, MON_T := T#20s, MON_T_STOP := T#20s, MPS := #"P-08.01".QDrive_Fault, L_FLOW_MON :=, FLOW :=, FLOW_LL :=, FLOW_MT :=, IN_SP_Speed :=, IN_SW := "P-08.01 SW", "IN _AV" := "P-08.01 AV", IN_Volt := "P-08.01 Voltage", IN_Ampere := "P-08.01 Ampere", IN_KW := "P-08.01 KW", IN_Nm := "P-08.01 Nm", INSTANCE := 'P-08.01', RESTART :=, VISIBILITY :=, OPdwCmd :=, QdwState =>, QwState =>, QSTOPPING =>, QSTOP =>, QSTARTING =>, QRUN =>, QCMD_ON =>, QMON =>, QMON_ERR =>, QMON_T =>, QMON_T_STOP =>, QFLOW_MON =>, QFLOW_MT =>, QFLOW_ERR =>, QMPS =>, QMAN_AUT =>, QREMOTE =>, QSIM =>, QLOCK =>, QERR =>, QERR_EXT =>, QDrive_Fault =>, QDrive_Alarm =>, QwAlarm =>, Q_CW => "P-08.01 CW", Q_SP_Speed => "P-08.01 SP", QAct_Speed =>, QAct_Volt =>, QAct_Amp =>, QAct_KW =>, QAct_Nm =>)
   END_RUNG
   RUNG wire#powerrail
      Contact( #lock )
   END_RUNG wire#w1
   RUNG wire#powerrail
      I_Contact( "DRP-P08.01" )
   END_RUNG wire#w1
   RUNG wire#powerrail
      I_Contact( #EM_Stop )
   END_RUNG wire#w2
   // the same network as SCL:
   #"P-08.01"(LOCK := #lock OR NOT "DRP-P08.01",   // "Motor_w_VSD"
              ERR_EXTERN := NOT #EM_Stop,
              LIOP_SEL := #Init,
              L_AUT := #Init,
              L_REMOTE := #Init,
              L_RESET := #Reset,
              L_MON := #Init,
              MON_T := T#20s,
              MON_T_STOP := T#20s,
              MPS := #"P-08.01".QDrive_Fault,
              IN_SW := "P-08.01 SW",
              "IN _AV" := "P-08.01 AV",
              IN_Volt := "P-08.01 Voltage",
              IN_Ampere := "P-08.01 Ampere",
              IN_KW := "P-08.01 KW",
              IN_Nm := "P-08.01 Nm",
              INSTANCE := 'P-08.01',
              Q_CW => "P-08.01 CW",
              Q_SP_Speed => "P-08.01 SP");
END_REGION

REGION Network 13: P-08.02
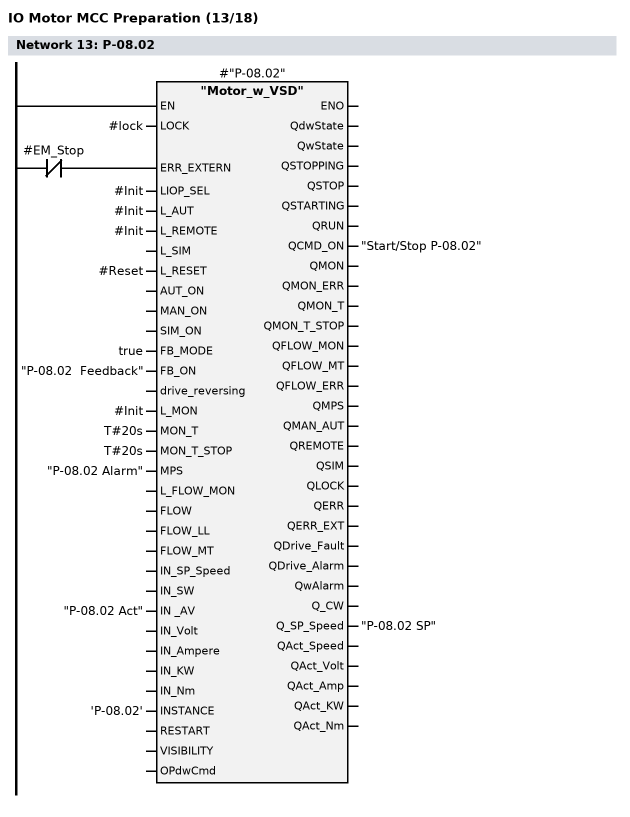
   RUNG wire#powerrail
      #"P-08.02"(ERR_EXTERN := wire#w1, LOCK := #lock, LIOP_SEL := #Init, L_AUT := #Init, L_REMOTE := #Init, L_SIM :=, L_RESET := #Reset, AUT_ON :=, MAN_ON :=, SIM_ON :=, FB_MODE := true, FB_ON := "P-08.02  Feedback", drive_reversing :=, L_MON := #Init, MON_T := T#20s, MON_T_STOP := T#20s, MPS := "P-08.02 Alarm", L_FLOW_MON :=, FLOW :=, FLOW_LL :=, FLOW_MT :=, IN_SP_Speed :=, IN_SW :=, "IN _AV" := "P-08.02 Act", IN_Volt :=, IN_Ampere :=, IN_KW :=, IN_Nm :=, INSTANCE := 'P-08.02', RESTART :=, VISIBILITY :=, OPdwCmd :=, QdwState =>, QwState =>, QSTOPPING =>, QSTOP =>, QSTARTING =>, QRUN =>, QCMD_ON => "Start/Stop P-08.02", QMON =>, QMON_ERR =>, QMON_T =>, QMON_T_STOP =>, QFLOW_MON =>, QFLOW_MT =>, QFLOW_ERR =>, QMPS =>, QMAN_AUT =>, QREMOTE =>, QSIM =>, QLOCK =>, QERR =>, QERR_EXT =>, QDrive_Fault =>, QDrive_Alarm =>, QwAlarm =>, Q_CW =>, Q_SP_Speed => "P-08.02 SP", QAct_Speed =>, QAct_Volt =>, QAct_Amp =>, QAct_KW =>, QAct_Nm =>)
   END_RUNG
   RUNG wire#powerrail
      I_Contact( #EM_Stop )
   END_RUNG wire#w1
   // the same network as SCL:
   #"P-08.02"(LOCK := #lock,   // "Motor_w_VSD"
              ERR_EXTERN := NOT #EM_Stop,
              LIOP_SEL := #Init,
              L_AUT := #Init,
              L_REMOTE := #Init,
              L_RESET := #Reset,
              FB_MODE := true,
              FB_ON := "P-08.02  Feedback",
              L_MON := #Init,
              MON_T := T#20s,
              MON_T_STOP := T#20s,
              MPS := "P-08.02 Alarm",
              "IN _AV" := "P-08.02 Act",
              INSTANCE := 'P-08.02',
              QCMD_ON => "Start/Stop P-08.02",
              Q_SP_Speed => "P-08.02 SP");
END_REGION

REGION Network 14: XA-09.01
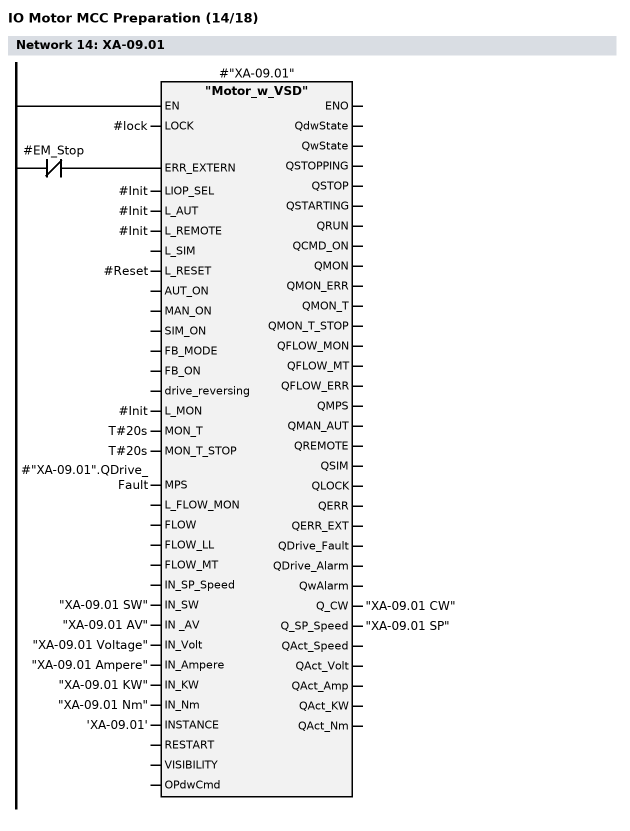
   RUNG wire#powerrail
      #"XA-09.01"(ERR_EXTERN := wire#w1, LOCK := #lock, LIOP_SEL := #Init, L_AUT := #Init, L_REMOTE := #Init, L_SIM :=, L_RESET := #Reset, AUT_ON :=, MAN_ON :=, SIM_ON :=, FB_MODE :=, FB_ON :=, drive_reversing :=, L_MON := #Init, MON_T := T#20s, MON_T_STOP := T#20s, MPS := #"XA-09.01".QDrive_Fault, L_FLOW_MON :=, FLOW :=, FLOW_LL :=, FLOW_MT :=, IN_SP_Speed :=, IN_SW := "XA-09.01 SW", "IN _AV" := "XA-09.01 AV", IN_Volt := "XA-09.01 Voltage", IN_Ampere := "XA-09.01 Ampere", IN_KW := "XA-09.01 KW", IN_Nm := "XA-09.01 Nm", INSTANCE := 'XA-09.01', RESTART :=, VISIBILITY :=, OPdwCmd :=, QdwState =>, QwState =>, QSTOPPING =>, QSTOP =>, QSTARTING =>, QRUN =>, QCMD_ON =>, QMON =>, QMON_ERR =>, QMON_T =>, QMON_T_STOP =>, QFLOW_MON =>, QFLOW_MT =>, QFLOW_ERR =>, QMPS =>, QMAN_AUT =>, QREMOTE =>, QSIM =>, QLOCK =>, QERR =>, QERR_EXT =>, QDrive_Fault =>, QDrive_Alarm =>, QwAlarm =>, Q_CW => "XA-09.01 CW", Q_SP_Speed => "XA-09.01 SP", QAct_Speed =>, QAct_Volt =>, QAct_Amp =>, QAct_KW =>, QAct_Nm =>)
   END_RUNG
   RUNG wire#powerrail
      I_Contact( #EM_Stop )
   END_RUNG wire#w1
   // the same network as SCL:
   #"XA-09.01"(LOCK := #lock,   // "Motor_w_VSD"
               ERR_EXTERN := NOT #EM_Stop,
               LIOP_SEL := #Init,
               L_AUT := #Init,
               L_REMOTE := #Init,
               L_RESET := #Reset,
               L_MON := #Init,
               MON_T := T#20s,
               MON_T_STOP := T#20s,
               MPS := #"XA-09.01".QDrive_Fault,
               IN_SW := "XA-09.01 SW",
               "IN _AV" := "XA-09.01 AV",
               IN_Volt := "XA-09.01 Voltage",
               IN_Ampere := "XA-09.01 Ampere",
               IN_KW := "XA-09.01 KW",
               IN_Nm := "XA-09.01 Nm",
               INSTANCE := 'XA-09.01',
               Q_CW => "XA-09.01 CW",
               Q_SP_Speed => "XA-09.01 SP");
END_REGION

REGION Network 15: P-09.01
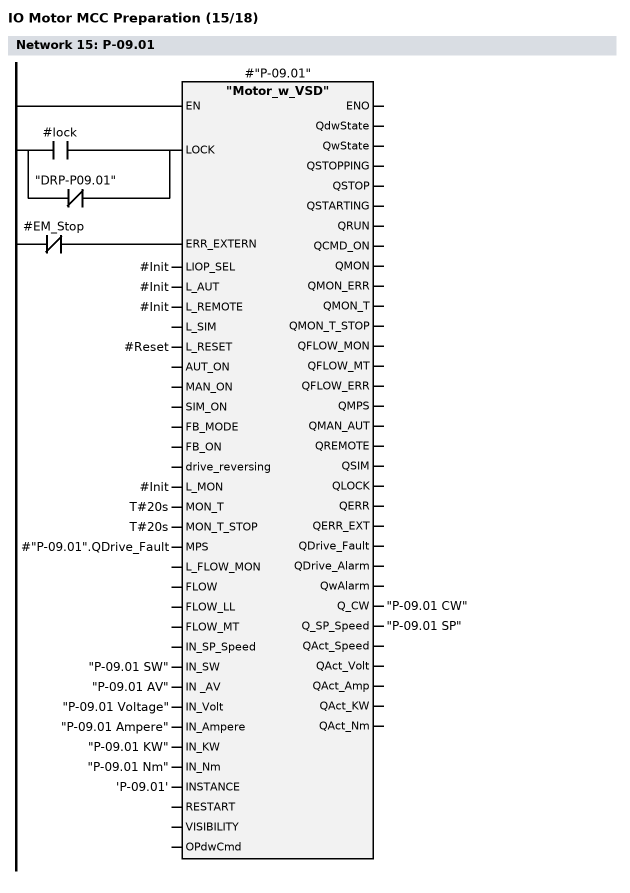
   RUNG wire#powerrail
      #"P-09.01"(LOCK := wire#w1, ERR_EXTERN := wire#w2, LIOP_SEL := #Init, L_AUT := #Init, L_REMOTE := #Init, L_SIM :=, L_RESET := #Reset, AUT_ON :=, MAN_ON :=, SIM_ON :=, FB_MODE :=, FB_ON :=, drive_reversing :=, L_MON := #Init, MON_T := T#20s, MON_T_STOP := T#20s, MPS := #"P-09.01".QDrive_Fault, L_FLOW_MON :=, FLOW :=, FLOW_LL :=, FLOW_MT :=, IN_SP_Speed :=, IN_SW := "P-09.01 SW", "IN _AV" := "P-09.01 AV", IN_Volt := "P-09.01 Voltage", IN_Ampere := "P-09.01 Ampere", IN_KW := "P-09.01 KW", IN_Nm := "P-09.01 Nm", INSTANCE := 'P-09.01', RESTART :=, VISIBILITY :=, OPdwCmd :=, QdwState =>, QwState =>, QSTOPPING =>, QSTOP =>, QSTARTING =>, QRUN =>, QCMD_ON =>, QMON =>, QMON_ERR =>, QMON_T =>, QMON_T_STOP =>, QFLOW_MON =>, QFLOW_MT =>, QFLOW_ERR =>, QMPS =>, QMAN_AUT =>, QREMOTE =>, QSIM =>, QLOCK =>, QERR =>, QERR_EXT =>, QDrive_Fault =>, QDrive_Alarm =>, QwAlarm =>, Q_CW => "P-09.01 CW", Q_SP_Speed => "P-09.01 SP", QAct_Speed =>, QAct_Volt =>, QAct_Amp =>, QAct_KW =>, QAct_Nm =>)
   END_RUNG
   RUNG wire#powerrail
      Contact( #lock )
   END_RUNG wire#w1
   RUNG wire#powerrail
      I_Contact( "DRP-P09.01" )
   END_RUNG wire#w1
   RUNG wire#powerrail
      I_Contact( #EM_Stop )
   END_RUNG wire#w2
   // the same network as SCL:
   #"P-09.01"(LOCK := #lock OR NOT "DRP-P09.01",   // "Motor_w_VSD"
              ERR_EXTERN := NOT #EM_Stop,
              LIOP_SEL := #Init,
              L_AUT := #Init,
              L_REMOTE := #Init,
              L_RESET := #Reset,
              L_MON := #Init,
              MON_T := T#20s,
              MON_T_STOP := T#20s,
              MPS := #"P-09.01".QDrive_Fault,
              IN_SW := "P-09.01 SW",
              "IN _AV" := "P-09.01 AV",
              IN_Volt := "P-09.01 Voltage",
              IN_Ampere := "P-09.01 Ampere",
              IN_KW := "P-09.01 KW",
              IN_Nm := "P-09.01 Nm",
              INSTANCE := 'P-09.01',
              Q_CW => "P-09.01 CW",
              Q_SP_Speed => "P-09.01 SP");
END_REGION

REGION Network 16: P-09.03 DOL
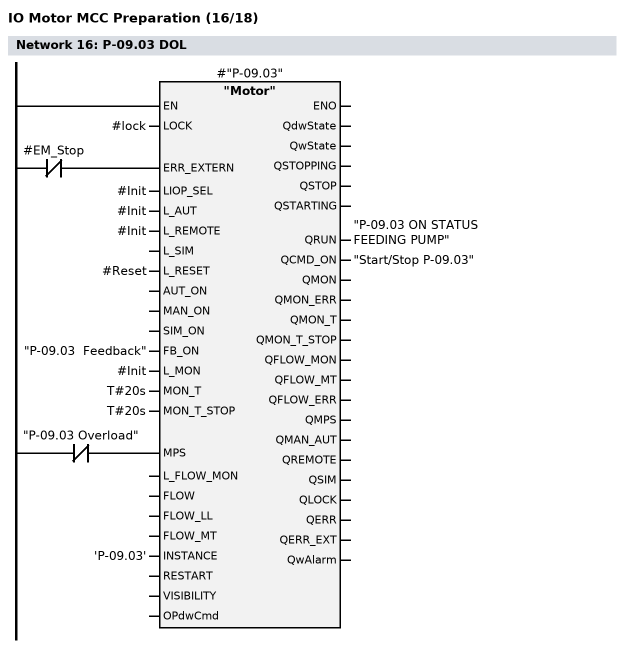
   RUNG wire#powerrail
      #"P-09.03"(ERR_EXTERN := wire#w1, MPS := wire#w2, LOCK := #lock, LIOP_SEL := #Init, L_AUT := #Init, L_REMOTE := #Init, L_SIM :=, L_RESET := #Reset, AUT_ON :=, MAN_ON :=, SIM_ON :=, FB_ON := "P-09.03  Feedback", L_MON := #Init, MON_T := T#20s, MON_T_STOP := T#20s, L_FLOW_MON :=, FLOW :=, FLOW_LL :=, FLOW_MT :=, INSTANCE := 'P-09.03', RESTART :=, VISIBILITY :=, OPdwCmd :=, QdwState =>, QwState =>, QSTOPPING =>, QSTOP =>, QSTARTING =>, QRUN => "P-09.03 ON STATUS FEEDING PUMP", QCMD_ON => "Start/Stop P-09.03", QMON =>, QMON_ERR =>, QMON_T =>, QMON_T_STOP =>, QFLOW_MON =>, QFLOW_MT =>, QFLOW_ERR =>, QMPS =>, QMAN_AUT =>, QREMOTE =>, QSIM =>, QLOCK =>, QERR =>, QERR_EXT =>, QwAlarm =>)
   END_RUNG
   RUNG wire#powerrail
      I_Contact( #EM_Stop )
   END_RUNG wire#w1
   RUNG wire#powerrail
      I_Contact( "P-09.03 Overload" )
   END_RUNG wire#w2
   // the same network as SCL:
   #"P-09.03"(LOCK := #lock,   // "Motor"
              ERR_EXTERN := NOT #EM_Stop,
              LIOP_SEL := #Init,
              L_AUT := #Init,
              L_REMOTE := #Init,
              L_RESET := #Reset,
              FB_ON := "P-09.03  Feedback",
              L_MON := #Init,
              MON_T := T#20s,
              MON_T_STOP := T#20s,
              MPS := NOT "P-09.03 Overload",
              INSTANCE := 'P-09.03',
              QRUN => "P-09.03 ON STATUS FEEDING PUMP",
              QCMD_ON => "Start/Stop P-09.03");
END_REGION

REGION Network 17: P-10.01
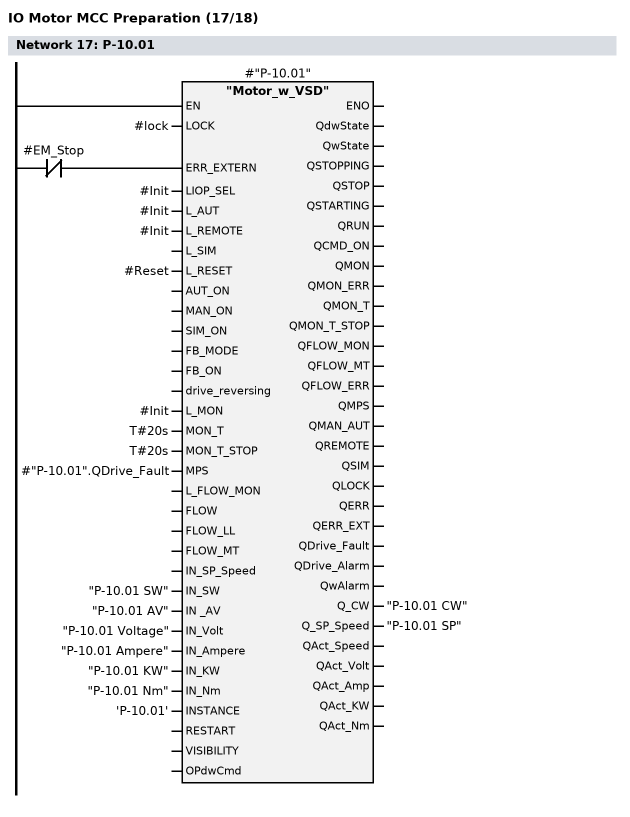
   RUNG wire#powerrail
      #"P-10.01"(ERR_EXTERN := wire#w1, LOCK := #lock, LIOP_SEL := #Init, L_AUT := #Init, L_REMOTE := #Init, L_SIM :=, L_RESET := #Reset, AUT_ON :=, MAN_ON :=, SIM_ON :=, FB_MODE :=, FB_ON :=, drive_reversing :=, L_MON := #Init, MON_T := T#20s, MON_T_STOP := T#20s, MPS := #"P-10.01".QDrive_Fault, L_FLOW_MON :=, FLOW :=, FLOW_LL :=, FLOW_MT :=, IN_SP_Speed :=, IN_SW := "P-10.01 SW", "IN _AV" := "P-10.01 AV", IN_Volt := "P-10.01 Voltage", IN_Ampere := "P-10.01 Ampere", IN_KW := "P-10.01 KW", IN_Nm := "P-10.01 Nm", INSTANCE := 'P-10.01', RESTART :=, VISIBILITY :=, OPdwCmd :=, QdwState =>, QwState =>, QSTOPPING =>, QSTOP =>, QSTARTING =>, QRUN =>, QCMD_ON =>, QMON =>, QMON_ERR =>, QMON_T =>, QMON_T_STOP =>, QFLOW_MON =>, QFLOW_MT =>, QFLOW_ERR =>, QMPS =>, QMAN_AUT =>, QREMOTE =>, QSIM =>, QLOCK =>, QERR =>, QERR_EXT =>, QDrive_Fault =>, QDrive_Alarm =>, QwAlarm =>, Q_CW => "P-10.01 CW", Q_SP_Speed => "P-10.01 SP", QAct_Speed =>, QAct_Volt =>, QAct_Amp =>, QAct_KW =>, QAct_Nm =>)
   END_RUNG
   RUNG wire#powerrail
      I_Contact( #EM_Stop )
   END_RUNG wire#w1
   // the same network as SCL:
   #"P-10.01"(LOCK := #lock,   // "Motor_w_VSD"
              ERR_EXTERN := NOT #EM_Stop,
              LIOP_SEL := #Init,
              L_AUT := #Init,
              L_REMOTE := #Init,
              L_RESET := #Reset,
              L_MON := #Init,
              MON_T := T#20s,
              MON_T_STOP := T#20s,
              MPS := #"P-10.01".QDrive_Fault,
              IN_SW := "P-10.01 SW",
              "IN _AV" := "P-10.01 AV",
              IN_Volt := "P-10.01 Voltage",
              IN_Ampere := "P-10.01 Ampere",
              IN_KW := "P-10.01 KW",
              IN_Nm := "P-10.01 Nm",
              INSTANCE := 'P-10.01',
              Q_CW => "P-10.01 CW",
              Q_SP_Speed => "P-10.01 SP");
END_REGION

REGION Network 18: P-51.01
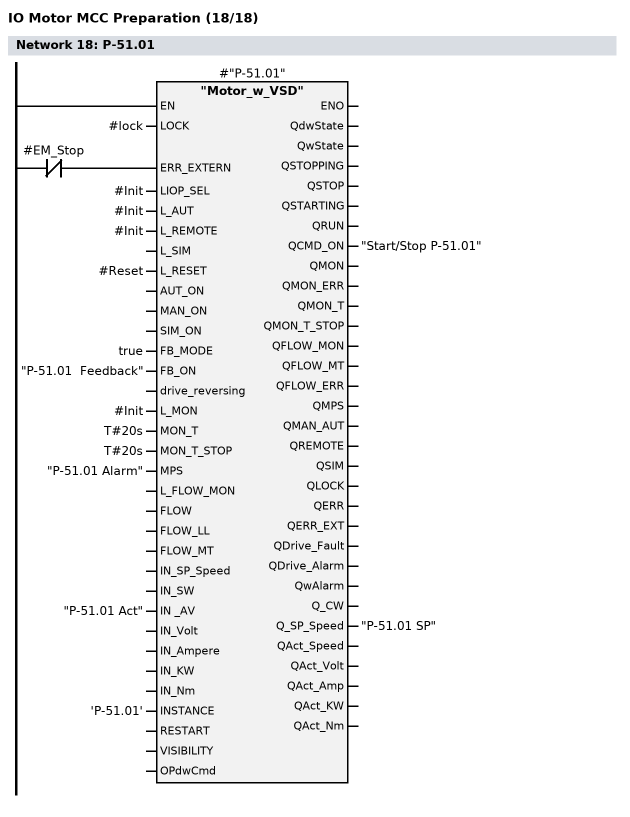
   RUNG wire#powerrail
      #"P-51.01"(ERR_EXTERN := wire#w1, LOCK := #lock, LIOP_SEL := #Init, L_AUT := #Init, L_REMOTE := #Init, L_SIM :=, L_RESET := #Reset, AUT_ON :=, MAN_ON :=, SIM_ON :=, FB_MODE := true, FB_ON := "P-51.01  Feedback", drive_reversing :=, L_MON := #Init, MON_T := T#20s, MON_T_STOP := T#20s, MPS := "P-51.01 Alarm", L_FLOW_MON :=, FLOW :=, FLOW_LL :=, FLOW_MT :=, IN_SP_Speed :=, IN_SW :=, "IN _AV" := "P-51.01 Act", IN_Volt :=, IN_Ampere :=, IN_KW :=, IN_Nm :=, INSTANCE := 'P-51.01', RESTART :=, VISIBILITY :=, OPdwCmd :=, QdwState =>, QwState =>, QSTOPPING =>, QSTOP =>, QSTARTING =>, QRUN =>, QCMD_ON => "Start/Stop P-51.01", QMON =>, QMON_ERR =>, QMON_T =>, QMON_T_STOP =>, QFLOW_MON =>, QFLOW_MT =>, QFLOW_ERR =>, QMPS =>, QMAN_AUT =>, QREMOTE =>, QSIM =>, QLOCK =>, QERR =>, QERR_EXT =>, QDrive_Fault =>, QDrive_Alarm =>, QwAlarm =>, Q_CW =>, Q_SP_Speed => "P-51.01 SP", QAct_Speed =>, QAct_Volt =>, QAct_Amp =>, QAct_KW =>, QAct_Nm =>)
   END_RUNG
   RUNG wire#powerrail
      I_Contact( #EM_Stop )
   END_RUNG wire#w1
   // the same network as SCL:
   #"P-51.01"(LOCK := #lock,   // "Motor_w_VSD"
              ERR_EXTERN := NOT #EM_Stop,
              LIOP_SEL := #Init,
              L_AUT := #Init,
              L_REMOTE := #Init,
              L_RESET := #Reset,
              FB_MODE := true,
              FB_ON := "P-51.01  Feedback",
              L_MON := #Init,
              MON_T := T#20s,
              MON_T_STOP := T#20s,
              MPS := "P-51.01 Alarm",
              "IN _AV" := "P-51.01 Act",
              INSTANCE := 'P-51.01',
              QCMD_ON => "Start/Stop P-51.01",
              Q_SP_Speed => "P-51.01 SP");
END_REGION
END_FUNCTION_BLOCK
